TYPE ST_BaseEvents_Memory :
STRUCT
	arrRow						: ARRAY [1..GVL_BaseConstans.MAX_EVENTS_IN_MEMORY] OF ST_BaseEvents_RowInMemory;
	iNumberOfRow				: INT;
	
END_STRUCT
END_TYPE

(* stored: Version 1.1.0.1
   DUT ST_BaseEvents_Memory: Id {089aa9a1-f075-03e9-310d-329f75ba9664} *)
